// TIA Portal V17 export
BLOCK "FC_Counters"   // ObjectSW13, LAD
BEGIN

REGION Network 1: ctu
END_REGION

REGION Network 2: ctd
END_REGION

REGION Network 3: ctud
END_REGION
END_BLOCK
